// TIA Portal V20 export
TYPE "typeFDoorUnlockOutput"
// stored: Access Published, IsFailsafeCompliant true, Namespace Safety
   STRUCT
      UnwinderTopDoorUnlock : Bool;   // F Door Unlock Cmd Status
      UnwinderLeftDoorUnlock : Bool;   // F Door Unlock Cmd Status
      UnwinderRightDoorUnlock : Bool;   // F Door Unlock Cmd Status
      CutterDoorUnlock : Bool;   // F Door Unlock Cmd Status
      MagazineDoorUnlock : Bool;   // F Door Unlock Cmd Status
      ConveyorDoorUnlock : Bool;   // F Door Unlock Cmd Status
      ScrapBoxDoorUnlock : Bool;   // F Door Unlock Cmd Status
      CentralAisleDoorUnlock : Bool;   // F Door Unlock Cmd Status
      TotalOneDoorUnlock : Bool;   // F Door Unlock Cmd Status
   END_STRUCT;
END_TYPE
